PROGRAM MAIN
VAR
END_VAR

END_PROGRAM

(* stored: Version 1.1.0.1, ProductVersion 3.1.4024.12
   POU MAIN: Id {4ad3dadb-4c25-4835-a240-c5ba522501df}, SpecialFunc None *)
